TYPE ByteReal :
UNION
	rValue : REAL;    // Needs 4 Bytes in memory
    abValue:  ARRAY [1..4] OF BYTE;
END_UNION
END_TYPE

(* stored: Version 1.1.0.1, ProductVersion 3.1.4022.18
   DUT ByteReal: Id {ee93410b-e195-4eac-a529-5c07e892c104} *)
